PROGRAM Structure_MAIN
VAR
	baseTime:TIME; //tempo universel à utiliser n'importe où avec la fonction delay()
END_VAR
VAR_INPUT
	IbStartInit: BOOL;
	IbStartMatch: BOOL;
	IbChoixCote: BOOL;
	IiChoixParcours: INT;
	IbMoteurOn:BOOL;
	IbPauseMotion : BOOL;
	IbEndMatch:BOOL;
	IbAbortTask:BOOL;
	IbPyScriptActive : BOOL;
	IiNumDynamixel:INT;
END_VAR
VAR_OUTPUT
	QbmoteurPower:BOOL;
	QbmoteurStop:BOOL;
	QbstartBalise:BOOL;
	QbMatchEnCours:BOOL;
	QbstartPyScript:BOOL;
	QbEtapeEnCours:STRING(50);
END_VAR
//TO DO
(*
1. Créer la séquence d'init
2. Gérer le choix de parcour dans le prématch
3. Modifier les actions en fonctions du tableau
4. Ajouter les tableaux
5. Gérer le tiemout
6. Gérer l'interrruption
7. Gérer la séquence de fin de match
*)

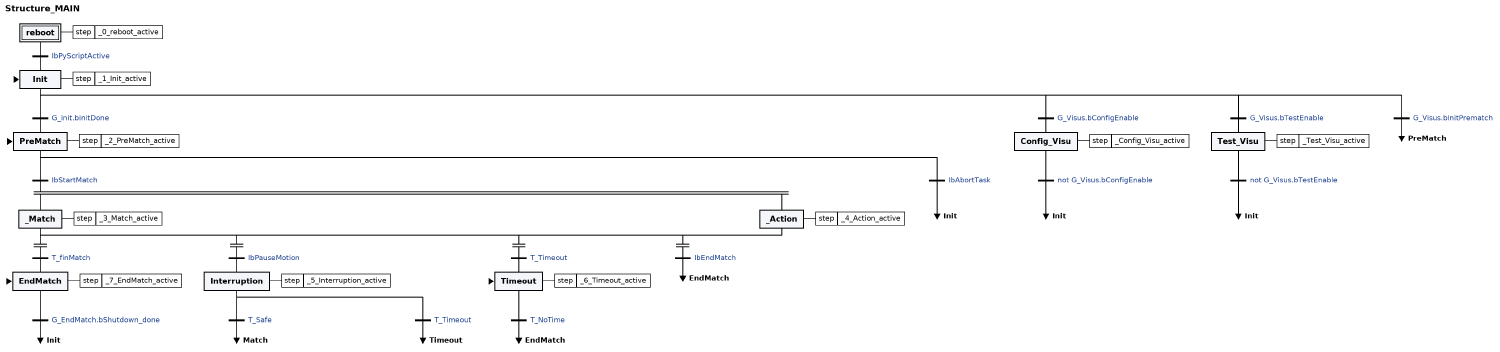
INITIAL_STEP reboot:
    _0_reboot_active(N);  // step action
END_STEP
TRANSITION FROM reboot TO Init
    := IbPyScriptActive;
END_TRANSITION
STEP Init:
    _1_Init_active(N);  // step action
END_STEP
TRANSITION FROM Init TO PreMatch
    := G_init.binitDone;
END_TRANSITION
TRANSITION FROM Init TO Config_Visu
    := G_Visus.bConfigEnable;
END_TRANSITION
STEP Config_Visu:
    _Config_Visu_active(N);  // step action
END_STEP
TRANSITION FROM Config_Visu TO Init
    := not G_Visus.bConfigEnable;
END_TRANSITION
TRANSITION FROM Init TO Test_Visu
    := G_Visus.bTestEnable;
END_TRANSITION
STEP Test_Visu:
    _Test_Visu_active(N);  // step action
END_STEP
TRANSITION FROM Test_Visu TO Init
    := not G_Visus.bTestEnable;
END_TRANSITION
TRANSITION FROM Init TO PreMatch
    := G_Visus.bInitPrematch;
END_TRANSITION
STEP PreMatch:
    _2_PreMatch_active(N);  // step action
END_STEP
TRANSITION FROM PreMatch TO (_Match, _Action)
    := IbStartMatch;
END_TRANSITION
TRANSITION FROM PreMatch TO Init
    := IbAbortTask;
END_TRANSITION
STEP _Match:
    _3_Match_active(N);  // step action
END_STEP
STEP _Action:
    _4_Action_active(N);  // step action
END_STEP
TRANSITION FROM (_Match, _Action) TO EndMatch
    := T_finMatch;
END_TRANSITION
STEP EndMatch:
    _7_EndMatch_active(N);  // step action
END_STEP
TRANSITION FROM EndMatch TO Init
    := G_EndMatch.bShutdown_done;
END_TRANSITION
TRANSITION FROM (_Match, _Action) TO Interruption
    := IbPauseMotion;
END_TRANSITION
STEP Interruption:
    _5_Interruption_active(N);  // step action
END_STEP
TRANSITION FROM Interruption TO (_Match, _Action)
    := T_Safe;
END_TRANSITION
TRANSITION FROM Interruption TO Timeout
    := T_Timeout;
END_TRANSITION
TRANSITION FROM (_Match, _Action) TO Timeout
    := T_Timeout;
END_TRANSITION
STEP Timeout:
    _6_Timeout_active(N);  // step action
END_STEP
TRANSITION FROM Timeout TO EndMatch
    := T_NoTime;
END_TRANSITION
TRANSITION FROM (_Match, _Action) TO EndMatch
    := IbEndMatch;
END_TRANSITION
// branch label Match

ACTION _0_reboot_active:
IF IbPyScriptActive THEN
	QbstartPyScript := FALSE;
ELSE
	QbstartPyScript := TRUE;
END_IF
END_ACTION

ACTION _1_Init_active:
IF IbAbortTask THEN
	G_init.ietapeInit := 0;
END_IF

CASE G_init.ietapeInit OF
	0://Mise à zéro et attende de l'ordre d'init
		QbstartBalise := FALSE;
		QbmoteurPower := FALSE;
		G_Prematch.bPrematchActive 	:= FALSE;
		G_EndMatch.bShutdown_done  	:= FALSE;
		G_Match.iLigne 				:= 0;
		IF IbStartInit THEN 
			G_init.ietapeInit := G_init.ietapeInit + 1;
		END_IF
	1://Mise sous tension des stepper moteurs de la base roulante (bloquage des roues)
		QbmoteurPower := TRUE;
		IF IbMoteurOn THEN
			G_init.ietapeInit := G_init.ietapeInit + 1;
			G_init.icounter := 1;
		END_IF;
	2://Activation du torque et des LED de tous les moteurs Dynamixels
		ITAction.DXLIN[G_init.icounter].bEnableTorque := TRUE;
		ITAction.DXLIN[G_init.icounter].bLedOn := TRUE;
		
		IF ITAction.DXLOUT[G_init.icounter].bEnableTorque AND ITAction.DXLOUT[G_init.icounter].bLedOn THEN 
			ITAction.DXLIN[G_init.icounter].bEnableTorque := FALSE;
			ITAction.DXLIN[G_init.icounter].bLedOn := FALSE;	
			G_init.icounter := G_init.icounter + 1;
		END_IF
		
		IF G_init.icounter > IiNumDynamixel THEN 
			G_init.ietapeInit := G_init.ietapeInit + 1;
		END_IF
		
	ELSE //Passage au prematch
		IF G_Visus.bInitPrematch OR G_Visus.bConfigEnable THEN 
			G_init.binitDone := TRUE;
			G_init.ietapeInit := 0;
		END_IF;
END_CASE

//à définir le nombre d'étape total pour que la visu affiche l'avancement sur une barre de progression
G_init.iNombreEtapeInit := 3;
G_Visus.iInitProgressBar := REAL_TO_INT(INT_TO_REAL(G_init.ietapeInit) / INT_TO_REAL(G_init.iNombreEtapeInit) * 100.0);

//switch en mode Test
IF VisuElems.CURRENTVISU = 'V_Test' THEN
	G_Visus.bTestEnable := TRUE;
ELSE
	G_Visus.bTestEnable := FALSE;
END_IF
END_ACTION

ACTION _2_PreMatch_active:
CASE IiChoixParcours OF
	0:
		P_Tableau_Strategie_1(bChoixCote := IbChoixCote);
		G_Match.Tableau := P_Tableau_Strategie_1.Tableau;
	1:
		P_Tableau_Strategie_2(bChoixCote := IbChoixCote);
		G_Match.Tableau := P_Tableau_Strategie_2.Tableau;
END_CASE

G_init.binitDone 			:= FALSE;
G_Match.PointMatch 			:= 0;
QbstartBalise 				:= FALSE;
G_Prematch.bPrematchActive 	:= TRUE;
ITMotion.odometrie.M_init_coordonne(IbChoixCote);
END_ACTION

ACTION _3_Match_active:
VisuElems.CURRENTVISU := 'V_Match';
//______________________________________________________________________________________________________________________________________________
//
// Comptage du Temps du match
//______________________________________________________________________________________________________________________________________________
IF NOT G_Match.MatchEnCours THEN
	G_Prematch.bPrematchActive := FALSE;
	G_Match.MatchEnCours := TRUE;
	G_Match.TimeStartMatch := TIME();
	G_Match.TimeStartLigne := TIME();
END_IF
G_Match.TimeMatch := TIME() - G_Match.TimeStartMatch; 

//______________________________________________________________________________________________________________________________________________
//
// Interpretation du Tableau
//______________________________________________________________________________________________________________________________________________
CASE G_Match.Tableau[G_Match.iLigne].TypeTache OF 
	

	//Temporisation-----------------------------------------------------------------------------------------------------------------------------
	eAttendre:
		IF delay(G_Match.TimeStartLigne, G_Match.Tableau[G_Match.iLigne].tAttente_ms)	THEN //Ligne suivante
			G_Match.PointMatch := G_Match.PointMatch + G_Match.Tableau[G_Match.iLigne].uiAjoutPoints_pts;
			G_Match.NextLigne := TRUE;
		END_IF
		
	//Change la ligne du Tableau-------------------------------------------------------------------------------------------------------------
	eChangementTache:
		FOR G_Match.iCounter := 1 TO 100 DO
			IF G_Match.Tableau[G_Match.iCounter].NomEtape = G_Match.Tableau[G_Match.iLigne].EtapeCible THEN
				G_Match.iLigne := G_Match.iCounter - 1;
				EXIT;
			END_IF
		END_FOR
		G_Match.NextLigne := TRUE;
	
	//Action du robot => se gère dans _4_Action_active-------------------------------------------------------------------------------------
	eAction: 
		IF G_Match.bActionFinie THEN //Ligne suivante
			G_Match.PointMatch := G_Match.PointMatch + G_Match.Tableau[G_Match.iLigne].uiAjoutPoints_pts;
			G_Match.NextLigne := TRUE;
		END_IF;	
	
	//Deplacement du robot-----------------------------------------------------------------------------------------------------------------------
	eDeplacement: 
		G_Match.bExecuteDeplacement := TRUE;
		IF G_Match.bDeplacementFini THEN //Ligne suivante
			G_Match.PointMatch := G_Match.PointMatch + G_Match.Tableau[G_Match.iLigne].uiAjoutPoints_pts;
			G_Match.bExecuteDeplacement := FALSE;
			G_Match.NextLigne := TRUE;
		END_IF
		
		//Gère le type de déplacement-------------------------------------------------------------------------------------------------------------
		CASE G_Match.Tableau[G_Match.iLigne].TypeDeplacement OF
			eCoordonne: 
				ITMotion.odometrie.M_move_to_coordonne(
				x 			:= G_Match.Tableau[G_Match.iLigne].lrPositionX_mm,
				y 			:= G_Match.Tableau[G_Match.iLigne].lrPositionY_mm,
				lrSpeed 	:= G_Match.Tableau[G_Match.iLigne].lrVitesse_mms,
				bExecute 	:= G_Match.bExecuteDeplacement,
				bbackward	:= FALSE,
				bDone 		=> G_Match.bDeplacementFini);
								
			eMarcheArriereCoordonne:
				ITMotion.odometrie.M_move_to_coordonne(
				x 			:= G_Match.Tableau[G_Match.iLigne].lrPositionX_mm,
				y 			:= G_Match.Tableau[G_Match.iLigne].lrPositionY_mm,
				lrSpeed 	:= G_Match.Tableau[G_Match.iLigne].lrVitesse_mms,
				bExecute 	:= G_Match.bExecuteDeplacement,
				bbackward	:= TRUE,
				bDone 		=> G_Match.bDeplacementFini);
			
			eDistance: 
				ITMotion.odometrie.M_move_distance(
				lrDistance 	:= G_Match.Tableau[G_Match.iLigne].lrDistanceVoulu_mm,
				lrSpeed 	:= G_Match.Tableau[G_Match.iLigne].lrVitesse_mms,
				bExecute 	:= G_Match.bExecuteDeplacement,
				bDone 		=> G_Match.bDeplacementFini);
				
			eAngle:
				ITMotion.odometrie.M_move_rotation(
				lrAngle 	:= G_Match.Tableau[G_Match.iLigne].lrAngleVoulu_deg,
				lrSpeed 	:= G_Match.Tableau[G_Match.iLigne].lrVitesse_mms,
				bExecute 	:= G_Match.bExecuteDeplacement,
				bDone 		=> G_Match.bDeplacementFini); 
			
			eCourbe:
				ITMotion.odometrie.M_move_curve(
				LrRayon		:= G_Match.Tableau[G_Match.iLigne].lrRayonCourbe_mm,
				LrAngle 	:= G_Match.Tableau[G_Match.iLigne].lrAngleVoulu_deg,
				lrSpeed 	:= G_Match.Tableau[G_Match.iLigne].lrVitesse_mms,				
				bExecute 	:= G_Match.bExecuteDeplacement,
				bDone 		=> G_Match.bDeplacementFini);
		END_CASE
END_CASE

//______________________________________________________________________________________________________________________________________________
//
// Passe à la ligne suivante du Tableau
//______________________________________________________________________________________________________________________________________________
IF G_Match.NextLigne THEN 
	G_Match.bActionFinie := FALSE;
	G_Match.bDeplacementFini := FALSE;
	G_Match.NextLigne := FALSE;
	G_Match.TimeStartLigne := TIME();
	G_Match.iLigne := G_Match.iLigne + 1; 
END_IF

//______________________________________________________________________________________________________________________________________________
//
// Debug
//______________________________________________________________________________________________________________________________________________

//affiche le nom de l'étape en cours pour le debug
IF G_Match.Tableau[G_Match.iLigne].NomEtape = '' THEN 
	QbEtapeEnCours := INT_TO_STRING(G_Match.iLigne); 
ELSE 
	QbEtapeEnCours := G_Match.Tableau[G_Match.iLigne].NomEtape;
END_IF;
END_ACTION

ACTION _4_Action_active:
IF G_Match.Tableau[G_Match.iLigne].TypeTache = eAction OR G_MAtch.iAsyncAction <> '' THEN 
///////////////////////////////////////////////////////////////////////////////////////////////////////////////////
// GESTION DES ACTIONS 
///////////////////////////////////////////////////////////////////////////////////////////////////////////////////

	IF StartAction('Lampe 3s') THEN
		
		G_IO.bLEDInit := TRUE;
		
		IF delay(G_match.TimeStartLigne, T#3S) THEN
			G_IO.bLEDInit := FALSE;
			FinishAction(0);
		END_IF;
		
//__________________________________________________________________________________________________________________
///////////////////////////////////////////////////////////////////////////////////////////////////////////////////
	ELSIF StartAction('Dynamixel position 0') THEN
		F_DXL_Position(0,500,ITAction.Template_XL);
//__________________________________________________________________________________________________________________
///////////////////////////////////////////////////////////////////////////////////////////////////////////////////		
	ELSIF StartAction('Dynamixel position 4095') THEN
		CASE G_Match.iEtapeAction OF
			0:
				ITAction.DXLIN[ITAction.Template_XL].bPosition := TRUE;
				ITAction.DXLIN[ITAction.Template_XL].ParamPosition_DINT := 10000;
				ITAction.DXLIN[ITAction.Template_XL].ParamSpeed_INT := 500;
				IF ITAction.DXLOUT[ITAction.Template_XL].bPosition THEN
					ITAction.DXLIN[ITAction.Template_XL].bPosition := FALSE;
					FinishAction(1);
					Next();
				END_IF
			1:
				ITAction.DXLIN[ITAction.Template_XL].bGetPosition := TRUE;
				IF PlusOuMoins(ITAction.DXLOUT[ITAction.Template_XL].INFO_Position_dint, 10000, 15) THEN 
					ITAction.DXLIN[ITAction.Template_XL].bGetPosition := FALSE;
					FinishAction(0);
				END_IF
		END_CASE
		
//__________________________________________________________________________________________________________________
///////////////////////////////////////////////////////////////////////////////////////////////////////////////////		
	ELSIF StartAction('Dynamixel reset') THEN
		F_DXL_Reset(ITAction.XLID2,1);
		
		
//__________________________________________________________________________________________________________________
///////////////////////////////////////////////////////////////////////////////////////////////////////////////////		
//--> Insérer les templates à partir d'ici 


///////////////////////////////////////////////////////////////////////////////////////////////////////////////////
// END_ACTION 
///////////////////////////////////////////////////////////////////////////////////////////////////////////////////
	ELSE //si aucune actione ne correspond au tableau TO DO
		pass();
	END_IF
END_IF



///////////////////////////////////////////////////////////////////////////////////////////////////////////////////
// DOCUMENTATION
///////////////////////////////////////////////////////////////////////////////////////////////////////////////////
(*

StartAction(Nom := "Nom de l'action");

FinishAction (StartAsync := FALSE, StopAsync := FALSE);

Next();

delay(last_time := G_Match.TimeStartLigne, tempo := T#1s);

PlusOuMoins(	val1  := G_A.DXL[G_A.Template].InfoPosition_DINT,
				val2  := 4095,
				plage := 15);
				
pass();
*)


///////////////////////////////////////////////////////////////////////////////////////////////////////////////////
// TEMPLATES A CUSTOMISER
///////////////////////////////////////////////////////////////////////////////////////////////////////////////////
(*
___________________________________________________________________________________________________________________

-> ACTION SIMPLE

///////////////////////////////////////////////////////////////////////////////////////////////////////////////////
	ELSIF StartAction('Nom Action') THEN
	
		"TON ACTION"
	
		IF "FIN DE L'ACTION" THEN
			FinishAction(0,0);
		END_IF
____________________________________________________________________________________________________________________		
		
-> CASE POUR L'ACTION

///////////////////////////////////////////////////////////////////////////////////////////////////////////////////
	ELSIF StartAction('Nom Action') THEN
		CASE G_Match.iEtapeAction OF
			0:
				IF "CONDITION POUR L'ETAPE SUIVANTE" THEN
					Next(); //etape suivante
				END_IF
			1:
				IF "FIN DE L'ACTION" THEN
					FinishAction(0,0);
				END_IF
		END_CASE
____________________________________________________________________________________________________________________

-> CASE POUR UNE ACTION ASYNCHRONE AVEC LE TABLEAU 
continue la suite du Tableau et l'action en même temps. Si le tableau arrive à une autre action, 
l'action asynchrone est terminée avant de commencer la prochaine action

///////////////////////////////////////////////////////////////////////////////////////////////////////////////////
	ELSIF StartAction('Nom Action') THEN
		CASE G_Match.iEtapeAction OF
			0:
				G_Match.iEtapeAction := G_Match.iEtapeAction + 1;
			1:
				FinishAction(StartAsync := TRUE,0);
			2:
				FinishAction(0,StopAsync := TRUE);
		END_CASE
____________________________________________________________________________________________________________________
*)
END_ACTION

ACTION _5_Interruption_active:
ITMotion.odometrie.M_reset_moteurs();
END_ACTION

ACTION _6_Timeout_active:

END_ACTION

ACTION _7_EndMatch_active:
IF G_Match.MatchEnCours THEN
	FOR G_EndMatch.icounter := 1 TO IiNumDynamixel DO
		ITAction.DXLIN[G_EndMatch.icounter].bGetLoad 		:= FALSE;
		ITAction.DXLIN[G_EndMatch.icounter].bGetMovement 	:= FALSE;
		ITAction.DXLIN[G_EndMatch.icounter].bGetPosition 	:= FALSE;
	END_FOR
	QbMoteurStop := TRUE;
	G_Match.MatchEnCours 	:= FALSE;
	baseTime := TIME();
END_IF

IF delay(baseTime, T#0.5S)THEN
	QbMoteurStop 			:= FALSE;
	QbstartBalise 			:= FALSE;
	QbmoteurPower 			:= FALSE;
	VisuElems.CURRENTVISU 	:= 'V_Fin_Match';
	IF NOT IbStartMatch THEN
			G_EndMatch.bShutdown_done := TRUE;
	END_IF
END_IF;
END_ACTION

ACTION _Config_Visu_active:
IF G_Visus.bConfigEnable THEN 
	VisuElems.CURRENTVISU := 'V_Config';
	//Move robot
	ITMotion.odometrie.M_move_to_coordonne(
	x 			:= G_Visus.lrConfigPosX,
	y 			:= G_Visus.lrConfigPosY,
	lrSpeed 	:= G_Visus.lrConfigVitesse,
	bExecute 	:= G_Visus.bConfigStart,
	bbackward	:= G_Visus.bConfigMarcheArriere,
	bDone 		=> G_Visus.bConfigMoveDone);
	
	//set acceleration / deceleration
	IF G_Visus.lrConfigAcc <> 0 OR G_Visus.lrConfigDecc <> 0 THEN
		ITMotion.odometrie.M_set_acceleration(lrAcc := G_Visus.lrConfigAcc, lrDecc := G_Visus.lrConfigDecc);
	END_IF
	
	//balise on
	QbstartBalise := G_Visus.bConfigBalise;
	
	//moteur on
	QbmoteurPower := G_Visus.bConfigMoteurPower;
	
	//bouton reset
	IF G_Visus.bConfigReset THEN 
		ITMotion.odometrie.M_init_coordonne(bChoixCote := G_Visus.bConfigChoixCote);
	END_IF
	
	//erreur et pourcentage 
	G_Visus.lrConfigErreurX := ABS(G_odometrie.lrPositionX - G_Visus.lrConfigPosX);
	G_Visus.lrConfigErreurY := ABS(G_odometrie.lrPositionY - G_Visus.lrConfigPosY);
	G_Visus.lrConfigErreurX_Pourcent := ABS(G_Visus.lrConfigErreurX/G_odometrie.lrPositionX)*100;
	G_Visus.lrConfigErreurY_Pourcent := ABS(G_Visus.lrConfigErreurY/G_odometrie.lrPositionY)*100;

ELSE// désactivation du mode config
	
	//remise à 0 des valeurs
	QbstartBalise := FALSE;	
	QbmoteurPower := FALSE;
	G_Visus.lrConfigErreurX :=0 ;
	G_Visus.lrConfigErreurY := 0;
	G_Visus.lrConfigErreurX_Pourcent := 0;
	G_Visus.lrConfigErreurY_Pourcent := 0;
	G_Visus.bConfigStart := 0;
	
	//retour au menu
	VisuElems.CURRENTVISU := 'V_Menu';
END_IF

//On doit refaire un init après être sorti du mode config
G_init.binitDone := FALSE;

//mouvement prêt à être effectué
G_Visus.bConfigMoteurReady := IbMoteurOn;

//Indicateur pour dire que le robot est prêt à effectuer un déplacement
IF G_Visus.bConfigMoveDone THEN 
	G_Visus.bConfigStart := FALSE;
END_IF

IF G_Visus.bConfigMoteurReady AND (G_Visus.bConfigStart AND G_Visus.bConfigMoveDone OR NOT G_Visus.bConfigStart)THEN 
	G_Visus.bConfigReady := TRUE;
ELSE
	G_Visus.bConfigReady := FALSE;	
END_IF
END_ACTION

ACTION _Test_Visu_active:
//quitte le mode visu si on retourne au menu
IF VisuElems.CURRENTVISU = 'V_Test' THEN
	G_Visus.bTestEnable := TRUE;
ELSE
	G_Visus.bTestEnable := FALSE;
END_IF

//On doit refaire un init après être sorti du mode Test
G_init.binitDone := FALSE;

IF G_Visus.bTestEnable THEN 
	IF    G_Visus.sTestBouton1 THEN
		G_Match.Tableau[G_Match.iLigne].TypeAction := G_Visus.sTestFunction1;
	ELSIF G_Visus.sTestBouton2 THEN
		G_Match.Tableau[G_Match.iLigne].TypeAction := G_Visus.sTestFunction2;
	ELSIF G_Visus.sTestBouton3 THEN
		G_Match.Tableau[G_Match.iLigne].TypeAction := G_Visus.sTestFunction3;
	ELSIF G_Visus.sTestBouton4 THEN
		G_Match.Tableau[G_Match.iLigne].TypeAction := G_Visus.sTestFunction4;
	ELSIF G_Visus.sTestBouton5 THEN
		G_Match.Tableau[G_Match.iLigne].TypeAction := G_Visus.sTestFunction5;
	ELSIF G_Visus.sTestBouton6 THEN
		G_Match.Tableau[G_Match.iLigne].TypeAction := G_Visus.sTestFunction6;
	END_IF
	
	// TO DO !!!
	//Définir le nom des actions testées 
	G_Visus.sTestFunction1 := 'Dynamixel position 4095';
	G_Visus.sTestFunction2 := 'Dynamixel position 0';
	G_Visus.sTestFunction3 := 'None';
	G_Visus.sTestFunction4 := 'None';
	G_Visus.sTestFunction5 := 'None';
	G_Visus.sTestFunction6 := 'None';
	
	///////////////////////////////////////////////////////////////////////////////////////////////////////////////////
	// GESTION DES ACTIONS 
	///////////////////////////////////////////////////////////////////////////////////////////////////////////////////
	IF StartAction('Dynamixel position 4095') THEN
		CASE G_Match.iEtapeAction OF
			0:
				ITAction.DXLIN[ITAction.Template_XL].bPosition := TRUE;
				ITAction.DXLIN[ITAction.Template_XL].ParamPosition_DINT := 10000;
				ITAction.DXLIN[ITAction.Template_XL].ParamSpeed_INT := 500;
				IF ITAction.DXLOUT[ITAction.Template_XL].bPosition THEN
					ITAction.DXLIN[ITAction.Template_XL].bPosition := FALSE;
					Next();
				END_IF
			1:
				ITAction.DXLIN[ITAction.Template_XL].bGetPosition := TRUE;
				IF PlusOuMoins(ITAction.DXLOUT[ITAction.Template_XL].INFO_Position_dint, 10000, 15) THEN 
					ITAction.DXLIN[ITAction.Template_XL].bGetPosition := FALSE;
					FinishAction(0);
				END_IF
		END_CASE
	//__________________________________________________________________________________________________________________
	///////////////////////////////////////////////////////////////////////////////////////////////////////////////////			
	ELSIF StartAction('Dynamixel position 0') THEN
		CASE G_Match.iEtapeAction OF
			0:
				ITAction.DXLIN[ITAction.Template_XL].bPosition := TRUE;
				ITAction.DXLIN[ITAction.Template_XL].ParamPosition_DINT := 1;
				ITAction.DXLIN[ITAction.Template_XL].ParamSpeed_INT := 1030;
				IF ITAction.DXLOUT[ITAction.Template_XL].bPosition THEN
					ITAction.DXLIN[ITAction.Template_XL].bPosition := FALSE;
					FinishAction(1);
					Next();;
				END_IF
			1:
				ITAction.DXLIN[ITAction.Template_XL].bGetPosition := TRUE;
				IF PlusOuMoins(ITAction.DXLOUT[ITAction.Template_XL].INFO_Position_dint, 1, 15) THEN 
					ITAction.DXLIN[ITAction.Template_XL].bGetPosition := FALSE;
					FinishAction(0);
				END_IF
		END_CASE
	//__________________________________________________________________________________________________________________
	///////////////////////////////////////////////////////////////////////////////////////////////////////////////////	
	END_IF
	
	//Action terminée
	if G_Match.bActionFinie then
		G_Match.Tableau[G_Match.iLigne].TypeAction := '';
		G_Match.bActionFinie := FALSE;
		
		G_Visus.sTestBouton1 := FALSE;
		G_Visus.sTestBouton2 := FALSE;
		G_Visus.sTestBouton3 := FALSE;
		G_Visus.sTestBouton4 := FALSE;
		G_Visus.sTestBouton5 := FALSE;
		G_Visus.sTestBouton6 := FALSE;
	END_IF

ELSE// désactivation du mode Test
	//remise à 0 des valeurs
	G_Match.bActionFinie := FALSE;
	G_Match.Tableau[G_Match.iLigne].TypeAction := '';
	G_Visus.sTestBouton1 := FALSE;
	G_Visus.sTestBouton2 := FALSE;
	G_Visus.sTestBouton3 := FALSE;
	G_Visus.sTestBouton4 := FALSE;
	G_Visus.sTestBouton5 := FALSE;
	G_Visus.sTestBouton6 := FALSE;
END_IF
END_ACTION

TRANSITION T_finMatch:
G_Match.Tableau[G_Match.iLigne].TypeTache = eFinParcours;
END_TRANSITION

TRANSITION T_NoTime:
G_Match.TimeMatch >= T#100s
END_TRANSITION

TRANSITION T_Safe:
not IbPauseMotion
END_TRANSITION

TRANSITION T_Timeout:
G_Match.TimeMatch > T#94s
END_TRANSITION

END_PROGRAM

(* stored: Version 1.1.0.1, ProductVersion 3.1.4024.12
   POU Structure_MAIN: Id {1a98f4bc-f3fd-4f90-9fe8-131cb98ad463}, SpecialFunc None
   Folder Transition: Id {468b4c47-ad8b-41d1-9bf1-238b9c1e89c7}
   Action _0_reboot_active: Id {8783d701-14ae-4d12-aa35-71479119d2e8}
   Action _1_Init_active: Id {9e1e986a-4c3a-4bce-9480-25a2b02a2470}
   Action _2_PreMatch_active: Id {aab04f3a-f9f9-4ad0-9e13-09943ec613d0}
   Action _3_Match_active: Id {97a2fb9a-5a70-4d35-afaf-27f682b48bd7}
   Action _4_Action_active: Id {3dd52e8e-5ec3-41e5-ad1a-9a5afb7f9d70}
   Action _5_Interruption_active: Id {5237f1ca-c328-4e04-be91-0752ad04c9c2}
   Action _6_Timeout_active: Id {d9a547ba-ecae-433a-9e89-06fa06b46c37}
   Action _7_EndMatch_active: Id {fd59140a-a49d-4fe9-80c3-9a33bc765eb8}
   Action _Config_Visu_active: Id {2d690fb6-8d79-4449-b377-091a708aad19}
   Action _Test_Visu_active: Id {1940a0ee-5791-4abb-a449-0f5e3b956797}
   Transition T_finMatch: Id {6d552d9d-9de1-4920-b9ad-cfd0f56aadd6}
   Transition T_NoTime: Id {38a228c7-2f1c-4951-94c3-fbe3a0077b5b}
   Transition T_Safe: Id {34370999-aba4-43de-97d4-009c3ee2ab09}
   Transition T_Timeout: Id {166cb7ce-9d6c-4a26-9ad2-e6973f3a32b0} *)
